{attribute 'GeneratedUsingTerminal: EM7004-0000-0017'}
{attribute addProperty BoxType "EM7004-0000-0017"}
{attribute addProperty Id "InputAT %I*Input_97D1F31316"}
{attribute addProperty CRC "2558703128"}
{attribute addProperty Size "16"}
TYPE DI_Inputs_9882B618 :
STRUCT
	{attribute addProperty Name "Input"}
	Input AT %I* : Input_97D1F313;
END_STRUCT
END_TYPE

(* stored: Version 1.2.0.0, ProductVersion 3.1.4024.9
   DUT DI_Inputs_9882B618: Id {eb4d437d-f6c2-487a-97e1-3e2208f3ab71} *)
